{attribute 'qualified_only'}
{attribute 'strict'}
TYPE E_CAN_Effenco :
(
	enum_member := 0
);
END_TYPE

(* stored: Version 1.1.0.1, ProductVersion 3.1.4024.12
   DUT E_CAN_Effenco: Id {4b49ff1b-a182-4b5b-acfe-079fa21b4b2d} *)
